# EPICS autosave request: support/sscan/2-6-4/sscanApp/Db/saveData_settings.req
$(P)saveData_fileSystem
$(P)saveData_subDir
$(P)saveData_baseName
$(P)saveData_scanNumber
$(P)saveData_realTime1D
$(P)saveData_maxAllowedRetries
$(P)saveData_retryWaitInSecs
